PROGRAM INTERNAL P_Builder_Example
VAR
	bStart : BOOL;
	nLn1, nLn2 : T_Size;
	sValue1, sValue2 : STRING(255);
	pString  : POINTER TO STRING;
	fbString_Builder1,
	fbString_Builder2 : FB_String_Builder;
END_VAR

IF bStart THEN
	bStart := FALSE;
	fbString_Builder2
		.Append(' I hate cats.')
		.Get_Buffer(pString);
	
	fbString_Builder1
		.Clear()
		.Append(' I love cats.')
		.Append(' I love dogs.')
		.Append_Buffer(pString)
		.Trim_Whitespace(T_Whitespace_Location.Both)
		.Get_Length(Length => nLn1)
		.Replace('cats','dogs',TRUE)
		.Insert(nLn1, ' Anaconda! ')
		.Split(nLn1,100, fbString_Builder2.Append(' Tigers are cats.'))
		.Get_Length(Length => nLn1);
	
	sValue1 := fbString_Builder1.To_Upper_Case().Get_String();
	sValue2 := fbString_Builder2
				.To_Lower_Case()
			   	.Trim_Whitespace(T_Whitespace_Location.Both)
				.Get_String();
	
	nLn2 := Tc2_Standard.LEN(sValue1);
	__DELETE(pString);
	END_IF

END_PROGRAM

(* stored: Version 1.1.0.1, ProductVersion 3.1.4024.4
   POU P_Builder_Example: Id {2fdd4b37-7a62-43c0-8687-8617b0ce492e}, SpecialFunc None *)
